// Mitsubishi GX Works2 project: BookEX6_45 ExtendedClock   PLC: Q13UDV

// global labels: Global
VAR_GLOBAL
  bVar0 AT M5000 : BOOL;
  abArray0 AT M5010 : ARRAY [0..49] OF BOOL;
  sStr0 AT D5000 : STRING[199];
  sStr1 AT D5100 : STRING[199];
  sStr2 AT D5200 : STRING[199];
  sStr3 AT D5300 : STRING[199];
  sStr4 AT D5400 : STRING[199];
  sStr5 AT D5500 : STRING[199];
  sStr6 AT D5600 : STRING[199];
  sStr7 AT D5700 : STRING[199];
  sStr8 AT D5800 : STRING[199];
  sStr9 AT D5900 : STRING[199];
  iVar0 AT D4500 : INT;
  iVar1 AT D4501 : INT;
  iVar2 AT D4502 : INT;
  iVar3 AT D4503 : INT;
  iVar4 AT D4504 : INT;
  iVar5 AT D4505 : INT;
  iVar6 AT D4506 : INT;
  iVar7 AT D4507 : INT;
  iVar8 AT D4508 : INT;
  iVar9 AT D4509 : INT;
  dVar0 AT D4510 : DINT;
  dVar1 AT D4512 : DINT;
  dVar2 AT D4514 : DINT;
  dVar3 AT D4516 : DINT;
  dVar4 AT D4518 : DINT;
  dVar5 AT D4520 : DINT;
  dVar6 AT D4522 : DINT;
  dVar7 AT D4524 : DINT;
  dVar8 AT D4526 : DINT;
  dVar9 AT D4528 : DINT;
  wVar0 AT D4530 : WORD;
  wVar1 AT D4531 : WORD;
  wVar2 AT D4532 : WORD;
  wVar3 AT D4533 : WORD;
  wVar4 AT D4534 : WORD;
  wVar5 AT D4535 : WORD;
  wVar6 AT D4536 : WORD;
  wVar7 AT D4537 : WORD;
  wVar8 AT D4538 : WORD;
  wVar9 AT D4539 : WORD;
  dwVar0 AT D4540 : DWORD;
  dwVar1 AT D4542 : DWORD;
  dwVar2 AT D4544 : DWORD;
  dwVar3 AT D4546 : DWORD;
  dwVar4 AT D4548 : DWORD;
  dwVar5 AT D4550 : DWORD;
  dwVar6 AT D4552 : DWORD;
  dwVar7 AT D4554 : DWORD;
  dwVar8 AT D4556 : DWORD;
  dwVar9 AT D4558 : DWORD;
  fsVar0 AT D4560 : REAL;
  fsVar1 AT D4562 : REAL;
  fsVar2 AT D4564 : REAL;
  fsVar3 AT D4566 : REAL;
  fsVar4 AT D4568 : REAL;
  fsVar5 AT D4570 : REAL;
  fsVar6 AT D4572 : REAL;
  fsVar7 AT D4574 : REAL;
  fsVar8 AT D4576 : REAL;
  fsVar9 AT D4578 : REAL;
  fdVar0 AT D4580 : LREAL;
  tTime0 AT D4620 : TIME;
  tTime1 AT D4622 : TIME;
  tTime2 AT D4624 : TIME;
  tTime3 AT D4626 : TIME;
  tTime4 AT D4628 : TIME;
  tTime5 AT D4630 : TIME;
  tTime6 AT D4632 : TIME;
  tTime7 AT D4634 : TIME;
  tTime8 AT D4636 : TIME;
  tTime9 AT D4638 : TIME;
  tTime10 AT D4640 : TIME;
  bVar1 AT M5001 : BOOL;
  bVar2 AT M5002 : BOOL;
  bVar3 AT M5003 : BOOL;
  bVar4 AT M5004 : BOOL;
  bVar5 AT M5005 : BOOL;
  bVar6 AT M5006 : BOOL;
  bVar7 AT M5007 : BOOL;
  bVar8 AT M5008 : BOOL;
  bVar9 AT M5009 : BOOL;
  abArray1 AT M5060 : ARRAY [0..49] OF BOOL;
  abArray2 AT M5110 : ARRAY [0..49] OF BOOL;
  abArray3 AT M5160 : ARRAY [0..49] OF BOOL;
  abArray4 AT M5210 : ARRAY [0..49] OF BOOL;
  abArray5 AT M5260 : ARRAY [0..49] OF BOOL;
  abArray6 AT M5310 : ARRAY [0..49] OF BOOL;
  abArray7 AT M5360 : ARRAY [0..49] OF BOOL;
  abArray8 AT M5410 : ARRAY [0..49] OF BOOL;
  abArray9 AT M5460 : ARRAY [0..49] OF BOOL;
  fdVar1 AT D4584 : LREAL;
  fdVar2 AT D4588 : LREAL;
  fdVar3 AT D4592 : LREAL;
  fdVar4 AT D4596 : LREAL;
  fdVar5 AT D4600 : LREAL;
  fdVar6 AT D4604 : LREAL;
  fdVar7 AT D4608 : LREAL;
  fdVar8 AT D4612 : LREAL;
  fdVar9 AT D4616 : LREAL;
  afsPen0 AT D2000 : ARRAY [0..499] OF REAL;
  afsPen1 AT D3000 : ARRAY [0..499] OF REAL;
  adwD10 AT D10 : ARRAY [0..9] OF DWORD;
  awD10 AT D10 : ARRAY [0..19] OF WORD;
  abM10 AT M10 : ARRAY [0..19] OF BOOL;
  aiClock AT D40 : ARRAY [0..6] OF INT;
  aiClock1 AT D40 : ARRAY [0..7] OF INT;
END_VAR

// global labels: QPLCSpecial
VAR_GLOBAL
  sbGetTime AT SM213 : BOOL;
  sbOn AT SM400 : BOOL;
  sbOff AT SM401 : BOOL;
  sbOn1Time AT SM402 : BOOL;
  sbOff1Time AT SM403 : BOOL;
  sb5ms AT SM409 : BOOL;
  sdSwitch AT SD200 : INT;
  sdTime03 AT SD212 : INT;
  sdTime04 AT SD213 : INT;
  sdTime02 AT SD211 : INT;
  sdTime01 AT SD210 : INT;
  sdScanTime1 AT SD521 : INT;
  sdScanTimeMin1 AT SD525 : INT;
  sdScanTimeMin AT SD524 : INT;
  sdScanTimeMax1 AT SD527 : INT;
  sdScanTimeMax AT SD526 : INT;
  sbErrInfo2 AT SM16 : BOOL;
  sbErrInfo AT SM5 : BOOL;
  sbSelfError AT SM1 : BOOL;
  sbDiagError AT SM0 : BOOL;
  sbResetErr AT SM50 : BOOL;
  sbSetTime AT SM210 : BOOL;
  sbFuse AT SM60 : BOOL;
  sbOpError AT SM56 : BOOL;
  sbPowerDown AT SM53 : BOOL;
  sbBatLow AT SM52 : BOOL;
  sbBatLowL AT SM51 : BOOL;
  sbSTOP AT SM203 : BOOL;
  sbPAUSE AT SM204 : BOOL;
  sbNsec AT SM414 : BOOL;
  sb1000ms AT SM413 : BOOL;
  sb500ms AT SM412 : BOOL;
  sbNms AT SM415 : BOOL;
  sbUserClk4 AT SM424 : BOOL;
  sbUserClk3 AT SM423 : BOOL;
  sbUserClk2 AT SM422 : BOOL;
  sbUserClk1 AT SM421 : BOOL;
  sbUserClk0 AT SM420 : BOOL;
  sdBatLowL AT SD51 : INT;
  sdPLCErrInfo AT SD4 : INT;
  sdPLCErrDate2 AT SD3 : INT;
  sdPLCErrDate1 AT SD2 : INT;
  sdPLCErrDate0 AT SD1 : INT;
  sdPLCErrCode AT SD0 : INT;
  sdFuse AT SD60 : INT;
  sdPowerDown AT SD53 : INT;
  sdBatLow AT SD52 : INT;
  sdCPUSts AT SD203 : INT;
  sdLed AT SD201 : INT;
  sdScanTime AT SD520 : INT;
  sdCntNsec AT SD414 : INT;
  sdCnt1sec AT SD412 : INT;
  sdCntScan AT SD420 : INT;
  sdCntNms AT SD415 : INT;
  sb100ms AT SM411 : BOOL;
  sb50ms AT SM410 : BOOL;
  sdSckOpenComp AT SD1282 : WORD;
  sdSckOpenReq AT SD1284 : WORD;
  sdSckDataRx AT SD1286 : WORD;
  sdSckConn AT SD1288 : WORD;
END_VAR
// user libraries (not included): HMI

FUNCTION_BLOCK GetDayOfWeek
VAR_INPUT
  bEN : BOOL;
END_VAR
VAR_OUTPUT
  bENO : BOOL;
END_VAR
VAR_INPUT
  iYear : INT;
END_VAR
VAR_OUTPUT
  o_DayWeek : INT;
END_VAR
VAR
  Result : INT;
END_VAR
VAR_INPUT
  iMonth : INT;
  iDay : INT;
END_VAR
VAR
  iY : INT;
  iC : INT;
  iM : INT;
  iYear2 : INT;
END_VAR

bENO 	:= bEN;
IF NOT bEN THEN
	RETURN;
END_IF;
IF iMonth <= 2 THEN
	iYear2 := iYear - 1;
	iM := iMonth + 12;
ELSE
	iYear2 := iYear;
	iM := iMonth;
END_IF;
iC := iYear2 / 100; 
iY := iYear2 MOD 100;
Result := ( (21*iC)/4 +(5* iY)/4 + (13 * (iM+1)) / 5 +iDay - 1) MOD 7; 
o_DayWeek := Result;
END_FUNCTION_BLOCK

FUNCTION LeapYear
VAR
  bLeap4 : BOOL;
  bLeap100 : BOOL;
  bLeap400 : BOOL;
END_VAR
VAR_INPUT
  i_Year : INT;
END_VAR
VAR
  bLeap : BOOL;
END_VAR
;
bLeap := FALSE;
IF (i_Year MOD 4) = 0 THEN bLeap4 := TRUE; ELSE bLeap4 := FALSE; END_IF;
IF (i_Year MOD 100) = 0 THEN bLeap100 := TRUE; ELSE bLeap100 := FALSE; END_IF;
IF (i_Year MOD 400) = 0 THEN bLeap400 := TRUE; ELSE bLeap400 := FALSE; END_IF;
IF (bLeap4 AND NOT bLeap100) OR bLeap400 THEN bLeap := TRUE; END_IF;
LeapYear := bLeap;
END_FUNCTION

PROGRAM ExDateMinus
VAR
  s1Time : ARRAY [0..4] OF INT;
  s2Time : ARRAY [0..4] OF INT;
  dTime : ARRAY [0..4] OF INT;
  Mov4INT_1 : Mov4INT;
  Mov4INT_2 : Mov4INT;
  Mov4INT_3 : Mov4INT;
  Mov4INT_4 : Mov4INT;
  Mov4INT_5 : Mov4INT;
  Mov4INT_6 : Mov4INT;
  tmp1 : INT;
  tmp2 : INT;
  tmp3 : INT;
  tmp4 : INT;
END_VAR
(* structured ladder/FBD written out as ST: instructions are called as NAME(EN, inputs, outputs); _pN, _eN, _tN stand for wires *)
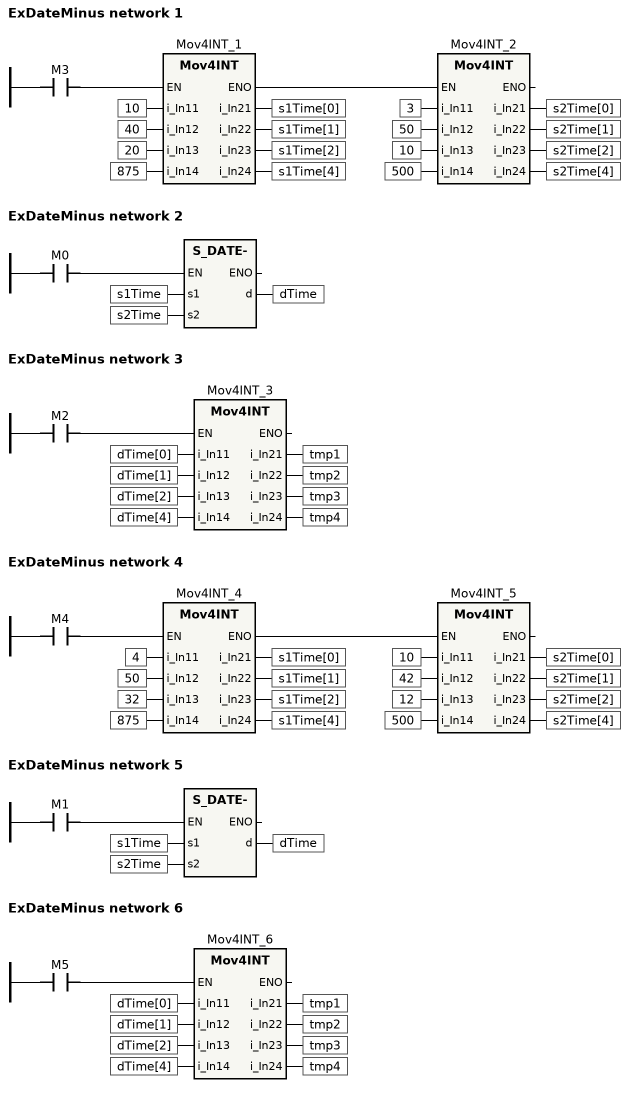
(* network 1 *)
Mov4INT_1(EN := M3, i_In11 := 10, i_In12 := 40, i_In13 := 20, i_In14 := 875, i_In21 => s1Time[0], i_In22 => s1Time[1], i_In23 => s1Time[2], i_In24 => s1Time[4]);
Mov4INT_2(EN := Mov4INT_1.ENO, i_In11 := 3, i_In12 := 50, i_In13 := 10, i_In14 := 500, i_In21 => s2Time[0], i_In22 => s2Time[1], i_In23 => s2Time[2], i_In24 => s2Time[4]);
(* network 2 *)
S_DATE-(M0, s1Time, s2Time, dTime);
(* network 3 *)
Mov4INT_3(EN := M2, i_In11 := dTime[0], i_In12 := dTime[1], i_In13 := dTime[2], i_In14 := dTime[4], i_In21 => tmp1, i_In22 => tmp2, i_In23 => tmp3, i_In24 => tmp4);
(* network 4 *)
Mov4INT_4(EN := M4, i_In11 := 4, i_In12 := 50, i_In13 := 32, i_In14 := 875, i_In21 => s1Time[0], i_In22 => s1Time[1], i_In23 => s1Time[2], i_In24 => s1Time[4]);
Mov4INT_5(EN := Mov4INT_4.ENO, i_In11 := 10, i_In12 := 42, i_In13 := 12, i_In14 := 500, i_In21 => s2Time[0], i_In22 => s2Time[1], i_In23 => s2Time[2], i_In24 => s2Time[4]);
(* network 5 *)
S_DATE-(M1, s1Time, s2Time, dTime);
(* network 6 *)
Mov4INT_6(EN := M5, i_In11 := dTime[0], i_In12 := dTime[1], i_In13 := dTime[2], i_In14 := dTime[4], i_In21 => tmp1, i_In22 => tmp2, i_In23 => tmp3, i_In24 => tmp4);
END_PROGRAM

PROGRAM ExDatePlus
VAR
  s1Time : ARRAY [0..4] OF INT;
  s2Time : ARRAY [0..4] OF INT;
  dTime : ARRAY [0..4] OF INT;
  Mov4INT_1 : Mov4INT;
  Mov4INT_2 : Mov4INT;
  Mov4INT_3 : Mov4INT;
  tmp1 : INT;
  tmp2 : INT;
  tmp3 : INT;
  tmp4 : INT;
  Mov4INT_4 : Mov4INT;
  Mov4INT_5 : Mov4INT;
  Mov4INT_6 : Mov4INT;
END_VAR
(* structured ladder/FBD written out as ST: instructions are called as NAME(EN, inputs, outputs); _pN, _eN, _tN stand for wires *)
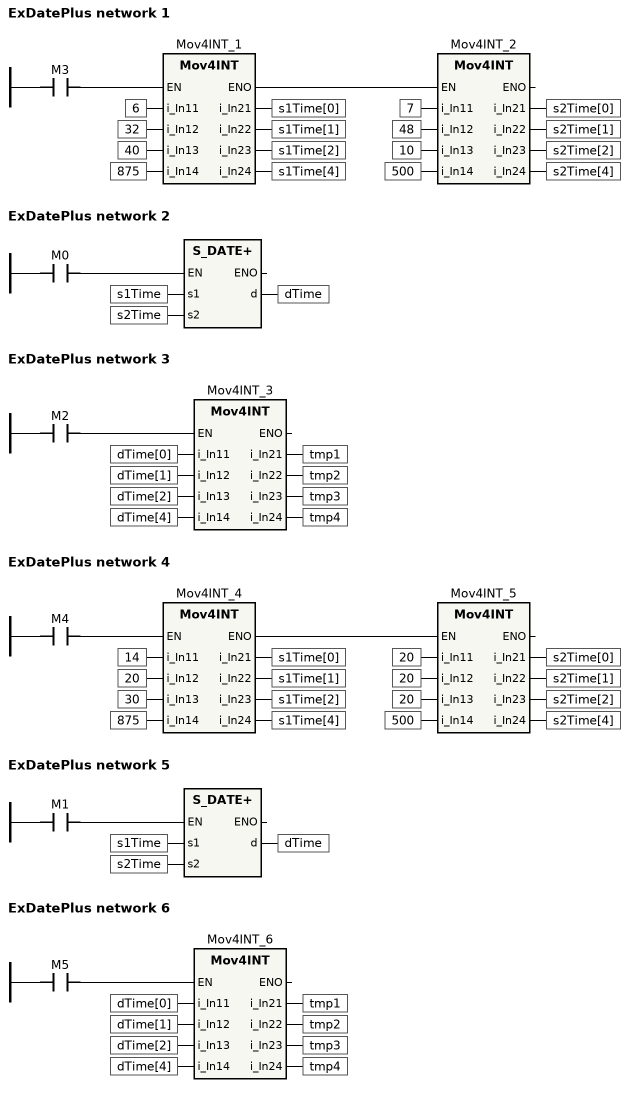
(* network 1 *)
Mov4INT_1(EN := M3, i_In11 := 6, i_In12 := 32, i_In13 := 40, i_In14 := 875, i_In21 => s1Time[0], i_In22 => s1Time[1], i_In23 => s1Time[2], i_In24 => s1Time[4]);
Mov4INT_2(EN := Mov4INT_1.ENO, i_In11 := 7, i_In12 := 48, i_In13 := 10, i_In14 := 500, i_In21 => s2Time[0], i_In22 => s2Time[1], i_In23 => s2Time[2], i_In24 => s2Time[4]);
(* network 2 *)
S_DATE+(M0, s1Time, s2Time, dTime);
(* network 3 *)
Mov4INT_3(EN := M2, i_In11 := dTime[0], i_In12 := dTime[1], i_In13 := dTime[2], i_In14 := dTime[4], i_In21 => tmp1, i_In22 => tmp2, i_In23 => tmp3, i_In24 => tmp4);
(* network 4 *)
Mov4INT_4(EN := M4, i_In11 := 14, i_In12 := 20, i_In13 := 30, i_In14 := 875, i_In21 => s1Time[0], i_In22 => s1Time[1], i_In23 => s1Time[2], i_In24 => s1Time[4]);
Mov4INT_5(EN := Mov4INT_4.ENO, i_In11 := 20, i_In12 := 20, i_In13 := 20, i_In14 := 500, i_In21 => s2Time[0], i_In22 => s2Time[1], i_In23 => s2Time[2], i_In24 => s2Time[4]);
(* network 5 *)
S_DATE+(M1, s1Time, s2Time, dTime);
(* network 6 *)
Mov4INT_6(EN := M5, i_In11 := dTime[0], i_In12 := dTime[1], i_In13 := dTime[2], i_In14 := dTime[4], i_In21 => tmp1, i_In22 => tmp2, i_In23 => tmp3, i_In24 => tmp4);
END_PROGRAM

PROGRAM ExDATERD
VAR
  Mov8INT2BCD_1 : Mov8INT2BCD;
  wBCD1 : WORD;
  wBCD2 : WORD;
  wBCD3 : WORD;
  wBCD4 : WORD;
  wBCD5 : WORD;
  wBCD6 : WORD;
  wBCD7 : WORD;
  wBCD8 : WORD;
  w2BCD1 : WORD;
  w2BCD2 : WORD;
  w2BCD3 : WORD;
  w2BCD4 : WORD;
  w2BCD5 : WORD;
  w2BCD6 : WORD;
  w2BCD7 : WORD;
  w2BCD8 : WORD;
END_VAR
(* structured ladder/FBD written out as ST: instructions are called as NAME(EN, inputs, outputs); _pN, _eN, _tN stand for wires *)
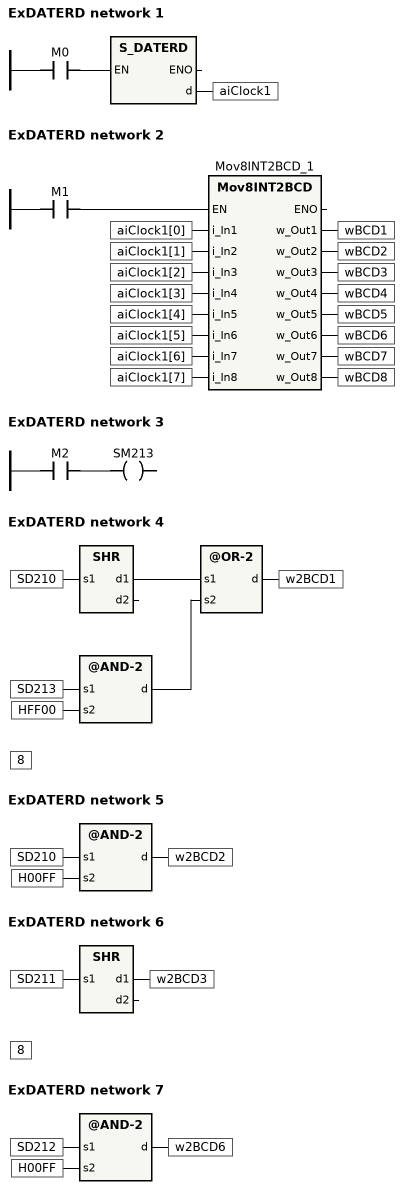
(* network 1 *)
S_DATERD(M0, aiClock1);
(* network 2 *)
Mov8INT2BCD_1(EN := M1, i_In1 := aiClock1[0], i_In2 := aiClock1[1], i_In3 := aiClock1[2], i_In4 := aiClock1[3], i_In5 := aiClock1[4], i_In6 := aiClock1[5], i_In7 := aiClock1[6], i_In8 := aiClock1[7], w_Out1 => wBCD1, w_Out2 => wBCD2, w_Out3 => wBCD3, w_Out4 => wBCD4, w_Out5 => wBCD5, w_Out6 => wBCD6, w_Out7 => wBCD7, w_Out8 => wBCD8);
(* network 3 *)
SM213 := M2;
(* network 4 *)
w2BCD1 := @OR-2(SHR(SD210), @AND-2(SD213, HFF00));
(* not connected to any output: 8 *)
(* network 5 *)
w2BCD2 := @AND-2(SD210, H00FF);
(* network 6 *)
w2BCD3 := SHR(SD211);
(* not connected to any output: 8 *)
(* network 7 *)
w2BCD6 := @AND-2(SD212, H00FF);
END_PROGRAM

PROGRAM ExGetDay
VAR
  GetDayOfWeek_1 : GetDayOfWeek;
END_VAR
(* structured ladder/FBD written out as ST: instructions are called as NAME(EN, inputs, outputs); _pN, _eN, _tN stand for wires *)
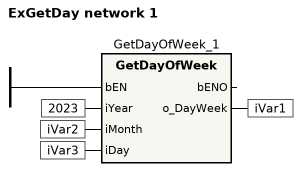
(* network 1 *)
GetDayOfWeek_1(bEN := TRUE, iYear := 2023, iMonth := iVar2, iDay := iVar3, o_DayWeek => iVar1);
END_PROGRAM

PROGRAM ExLeapYear
(* structured ladder/FBD written out as ST: instructions are called as NAME(EN, inputs, outputs); _pN, _eN, _tN stand for wires *)
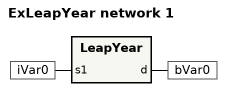
(* network 1 *)
bVar0 := LeapYear(iVar0);
END_PROGRAM
